TYPE ST_HeatStakeTemperatureSettings :
STRUCT
    // Nominal Heat Stake head operating window.
    rSetpointC              : LREAL := 215.0;
    rLowLimitC              : LREAL := 205.0;
    rHighLimitC             : LREAL := 225.0;
    rMaxTcDifferenceC       : LREAL := 10.0;

    tLowTemperatureTimeout  : TIME := T#5M;

    // Conservative initial tuning. FB_CTRL_PID is used with D disabled,
    // therefore the initial behaviour is PI.
    rKp                     : LREAL := 4.0;
    tTn                     : TIME := T#15S;
    tTv                     : TIME := T#0S;
    tTd                     : TIME := T#0S;

    tControllerCycle        : TIME := T#100MS;
    rOutputMinPercent       : LREAL := 0.0;
    rOutputMaxPercent       : LREAL := 100.0;

END_STRUCT
END_TYPE

(* stored: Version 1.1.0.1, ProductVersion 3.1.4026.18
   DUT ST_HeatStakeTemperatureSettings: Id {2907f69b-5179-4b5c-980d-9151f1af054e} *)
